PROGRAM MAIN
VAR
END_VAR

TrafficLight();

END_PROGRAM

(* stored: Version 1.1.0.1, ProductVersion 3.1.4024.12
   POU MAIN: Id {9cbfece7-1e67-454f-bff0-eecc8b7cd817}, SpecialFunc None *)
